// TIA Portal V20 export
FUNCTION_BLOCK "Simulation"   // FB101, LAD
// stored: MemoryReserve 100, Namespace Unit1.Em0, SetENOAutomatically false
   VAR
      Simulation_addon_Instance { S7_SetPoint := 'True'} : "Simulation_addon";
   END_VAR
BEGIN

REGION Network 1: cmExpelFwdBwd
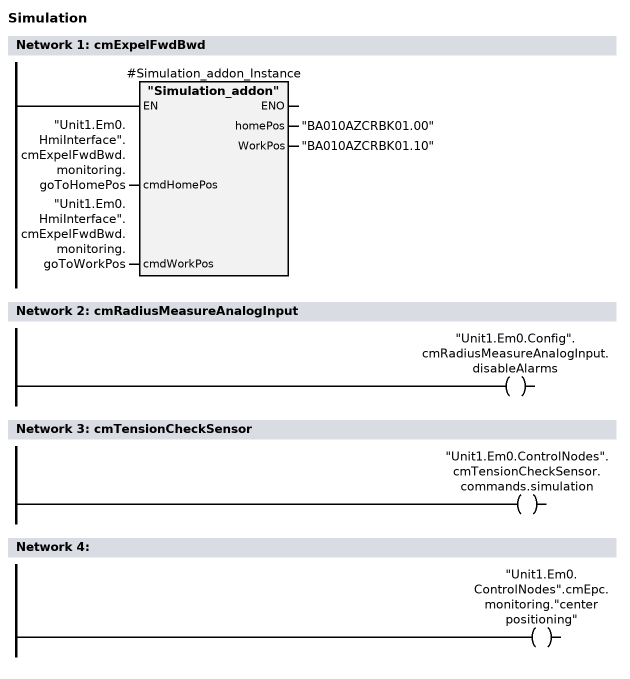
   RUNG wire#powerrail
      #Simulation_addon_Instance(cmdHomePos := "Unit1.Em0.HmiInterface".cmExpelFwdBwd.monitoring.goToHomePos, cmdWorkPos := "Unit1.Em0.HmiInterface".cmExpelFwdBwd.monitoring.goToWorkPos, homePos => "BA010AZCRBK01.00", WorkPos => "BA010AZCRBK01.10")
   END_RUNG
   // the same network as SCL:
   #Simulation_addon_Instance(cmdHomePos := "Unit1.Em0.HmiInterface".cmExpelFwdBwd.monitoring.goToHomePos,   // "Simulation_addon"
                           cmdWorkPos := "Unit1.Em0.HmiInterface".cmExpelFwdBwd.monitoring.goToWorkPos,
                           homePos => "BA010AZCRBK01.00",
                           WorkPos => "BA010AZCRBK01.10");
END_REGION

REGION Network 2: cmRadiusMeasureAnalogInput
   RUNG wire#powerrail
      Coil( "Unit1.Em0.Config".cmRadiusMeasureAnalogInput.disableAlarms )
   END_RUNG
   // the same network as SCL:
   "Unit1.Em0.Config".cmRadiusMeasureAnalogInput.disableAlarms := TRUE;
END_REGION

REGION Network 3: cmTensionCheckSensor
   RUNG wire#powerrail
      Coil( "Unit1.Em0.ControlNodes".cmTensionCheckSensor.commands.simulation )
   END_RUNG
   // the same network as SCL:
   "Unit1.Em0.ControlNodes".cmTensionCheckSensor.commands.simulation := TRUE;
END_REGION

REGION Network 4
   RUNG wire#powerrail
      Coil( "Unit1.Em0.ControlNodes".cmEpc.monitoring."center positioning" )
   END_RUNG
   // the same network as SCL:
   "Unit1.Em0.ControlNodes".cmEpc.monitoring."center positioning" := TRUE;
END_REGION
END_FUNCTION_BLOCK
